FUNCTION_BLOCK FB_Handoff EXTENDS FB_EquipmentModule_SR
VAR
    // Sub module definitions here

    // List of sub modules

    ipSubModules_Init : ARRAY[1..Parameters_PackML_Base.MAX_NO_OF_SUBMODULES] OF I_PackML_BaseModule := [];

    // Component definitions here

    CenteringClamp     : ARRAY[1..2] OF FB_DoubleSolenoidRetractFeedback := [(Name := 'Clamp_1'), (Name := 'Clamp_2')];
    BoardPresentSensor : FB_DigitalSensor                                := (Name := 'BoardPresentSensor');

    _ClampsClosed : BOOL;
END_VAR

VAR CONSTANT

    // Reports 

    FAULT : INT := 1;

    // Alarms

    PULL_WHEELS_ALARM_COUNT : INT := 5;
END_VAR

VAR
    _BoardDataToPass : ST_BoardData;
    _Location        : LREAL;
    _HoldingBoard    : BOOL;

    _ClampsOpen : BOOL;
END_VAR

PROPERTY ClampsClosed : bool
GET
ClampsClosed := _ClampsClosed;
END_GET
END_PROPERTY

PROPERTY ClampsOpen : bool
GET
ClampsOpen := _ClampsOpen;
END_GET
END_PROPERTY

METHOD CyclicLogic
VAR_INPUT
END_VAR
IF NOT _InitComplete THEN
    _InitComplete := Initialize();
    RETURN;
END_IF

SUPER^.CyclicLogic();

//HMI control for EM

fbControlSourceHMI.CyclicLogic();

//Set the current alarm severity for this module

// _CurrentAlarmSeverity := F_GetMaxSeverityRaised(Alarms:=PullWheelAlarms, CurrentSeverity:=_CurrentAlarmSeverity);

//Simulate Alarm Messaging

IF (CenteringClamp[1].InSimulation OR CenteringClamp[1].Retracted) AND (CenteringClamp[2].InSimulation OR CenteringClamp[2].Retracted) THEN
    _ClampsOpen := TRUE;
ELSE
    _ClampsOpen := FALSE;
END_IF

IF (CenteringClamp[1].InSimulation OR CenteringClamp[1].Extended) AND (CenteringClamp[2].InSimulation OR CenteringClamp[2].Extended) THEN
    _ClampsClosed := TRUE;
ELSE
    _ClampsClosed := FALSE;
END_IF

// CyclicLogicSimulation();
END_METHOD

PROPERTY DisableClamp1 : BOOL
SET
CenteringClamp[1].InSimulation := DisableClamp1;
END_SET
END_PROPERTY

PROPERTY DisableClamp2 : BOOL
SET
CenteringClamp[2].InSimulation := DisableClamp2;
END_SET
END_PROPERTY

METHOD GrabBoard : BOOL
VAR_INPUT
END_VAR
GrabBoard := FALSE;

FOR i := 1 TO 2 DO
    CenteringClamp[i].Extend();
END_FOR

IF CenteringClamp[1].Extended AND CenteringClamp[1].Extended THEN
    GrabBoard := TRUE;
    // 	Trace('Clamp Closed');
END_IF
END_METHOD

METHOD HMIControl
VAR_INPUT
END_VAR
IF HMI_INPUT[1] THEN
	FOR i := 1 TO 2 DO 
		ReleaseBoard(); 
	END_FOR
END_IF

IF HMI_INPUT[2] THEN
	FOR i := 1 TO 2 DO 
		GrabBoard(); 
	END_FOR
END_IF
END_METHOD

PROPERTY HoldingBoard : Bool
GET
HoldingBoard := _HoldingBoard;
END_GET
SET
_HoldingBoard := HoldingBoard;
END_SET
END_PROPERTY

//! @summary Basic module initialization logic
METHOD PROTECTED Initialize : BOOL;
VAR
    i                        : UDINT;
    varInfo                  : __SYSTEM.VAR_INFO;
    AllSubUnitsInitialized   : BOOL := TRUE;
    AllComponentsInitialized : BOOL := TRUE;
END_VAR

//! @description This method is called by <c>CyclicLogic()</c> as required
Initialize := FALSE;

CASE DescendantSequenceState OF
    0:
        RegisterComponent(BoardPresentSensor);

        FOR i := 1 TO 2 DO
            RegisterComponent(CenteringClamp[i]);
        END_FOR

        _LogModeChanges         := FALSE;
        _LogStateChanges        := FALSE;
        DescendantSequenceState := DescendantSequenceState + 10;

    10:
        //Setup Custom modes here

        (*CustomModes(eMode                          :=,
                    sName                          :=,
                    bDisableClearing               :=,
                    bDisableStarting               :=,
                    bDisableSuspended              :=,
                    bDisableStopping               :=,
                    bDisableAborting               :=,
                    bDisableHolding                :=,
                    bDisableHeld                   :=,
                    bDisableUnholding              :=,
                    bDisableSuspending             :=,
                    bDisableUnsuspending           :=,
                    bDisableResetting              :=,
                    bDisableIdle                   :=,
                    bDisableCompleting             :=,
                    bDisableComplete               :=,
                    bEnableUnitModeChangeStopped   :=,
                    bEnableUnitModeChangeIdle      :=,
                    bEnableUnitModeChangeSuspended :=,
                    bEnableUnitModeChangeExecute   :=,
                    bEnableUnitModeChangeAborted   :=,
                    bEnableUnitModeChangeHeld      :=,
                    bEnableUnitModeChangeComplete  :=,
                    bError                         =>,
                    nErrorId                       =>);*)

        DescendantSequenceState := DescendantSequenceState + 10;

    20:
        //Copy Mode names

        FOR i := 1 TO 3 DO
            ModeNames[i] := F_UnitModeToString(UDINT_TO_DINT(i));
        END_FOR

        RegisterExternalController(Controller := fbControlSourceHMI);
        fbControlSourceHMI.CyclicLogic();
        DescendantSequenceState := DescendantSequenceState + 10;

    30:
        //Call the Super

        IF SUPER^.Initialize() THEN
            DescendantSequenceState := DescendantSequenceState + 10;
        END_IF

    40:
        Initialize := TRUE;
END_CASE
END_METHOD

PROPERTY Location : LREAL
GET
Location := _Location;
END_GET
SET
_Location := Location;
END_SET
END_PROPERTY

METHOD ReleaseBoard : BOOL
VAR_INPUT
END_VAR
ReleaseBoard := FALSE;

FOR i := 1 TO 2 DO
    CenteringClamp[i].Retract();
END_FOR

IF CenteringClamp[1].Retracted AND CenteringClamp[1].Retracted THEN
    ReleaseBoard := TRUE;
    // 	Trace('Clamp Opened');
END_IF
END_METHOD

PROPERTY Request_WS : E_WaitSync
SET
_RequestedWaitSync := Request_WS;
END_SET
END_PROPERTY

PROPERTY Response_WS : E_WaitSync
GET
Response_WS := _ResponseWaitSync;
END_GET
END_PROPERTY

END_FUNCTION_BLOCK

(* stored: Version 1.1.0.1
   POU FB_Handoff: Id {70da996e-78d6-44ec-bec2-b5cc40f00560}, SpecialFunc None
   Folder I_CyclicFB: Id {60b30b9f-13bb-4d98-9723-a91813391450}
   Folder Methods: Id {7677dcc4-de99-4bb2-94de-30decda7f97c}
   Folder Properties: Id {fcb5a7db-9494-4a81-b51a-d5a8f8326cfd}
   Property ClampsClosed: Id {d62e2521-b6b0-4a38-83da-6d69cfbf9f62}
   Get Get: Id {e62dc733-dc06-402a-b106-887c215393d8}
   Property ClampsOpen: Id {d1dd4d10-0421-461d-93e4-d85eac30f7fe}
   Get Get: Id {26b61293-9d81-4ef0-a4ad-fef93cf56f94}
   Method CyclicLogic: Id {2a27383a-3bdf-4b88-9dfa-fe4625c84c7f}
   Property DisableClamp1: Id {f4898869-5589-495c-aac7-215a2e397a19}
   Set Set: Id {01c09bbf-070f-40d5-a327-10c5a0a3640c}
   Property DisableClamp2: Id {0f647c9a-201d-445d-b53d-a4c5cf5af2b3}
   Set Set: Id {7e84259a-0f94-4fd0-9325-8e0707dce915}
   Method GrabBoard: Id {30074c16-8805-4b76-8b9c-a185a15a2001}
   Method HMIControl: Id {7e2f3a4a-e0a7-47d0-befd-d576573fb5db}
   Property HoldingBoard: Id {bb7b46f1-f485-4aa9-b1e8-6b31ac586359}
   Get Get: Id {a88e5869-f233-4605-a2af-bbcad9d0432d}
   Set Set: Id {921ca532-95c2-494c-bd54-bec962bd8e85}
   Method Initialize: Id {ae611370-cb56-48df-8475-dd2b27dfd90a}
   Property Location: Id {edc54518-17de-47a8-a768-b0f44af3d18b}
   Get Get: Id {a82cde8e-973d-4022-b722-fd1c01e84813}
   Set Set: Id {4128df58-d7ea-4dfd-9927-fc63ffa4e234}
   Method ReleaseBoard: Id {53bbb63b-1d98-4640-9fed-58e0300cc527}
   Property Request_WS: Id {bbc4f125-8f63-48e8-9685-e90719f469bc}
   Set Set: Id {bdc578e3-a406-483d-91ae-b380bf1aeff0}
   Property Response_WS: Id {8b560b72-76e6-4e35-bf39-9ecbde73da2f}
   Get Get: Id {2f5b85e5-6a38-4e0e-a6fe-8959f5a35dc9} *)
